// TIA Portal V20 export
FUNCTION "ST002示教台" : Void   // FC3, LAD
{ S7_Optimized_Access := 'TRUE' }
// stored: SetENOAutomatically false
BEGIN

REGION Network 1
   // IW256 G120状态字
   // IW258 G120当前频率（16#0-16#4000,对应0-50hz)
   // QW256 G120控制字
   // QW258 G120当前频率（16#0-16#4000,对应0-50hz)
END_REGION
END_FUNCTION
